FUNCTION FC_InitRaInterface : BOOL
VAR_INPUT
END_VAR
VAR
	i: UINT;
	m_statesEnum: EProcessVariables;
END_VAR

// OUT - alarms
FOR i := ResiConst.ARR_MIN TO RaInterface_GVL.ALARM_ARR_MAX DO
	RaInterface_GVL.Out_Alarms[i].Active := FALSE;
	RaInterface_GVL.Out_Alarms[i].AlarmId := 0;
	RaInterface_GVL.Out_Alarms[i].InstanceName := '';
	RaInterface_GVL.Out_Alarms[i].Message := '';
	RaInterface_GVL.Out_Alarms[i].Severity := ESeverity.none;
	RaInterface_GVL.Out_Alarms[i].TimeTicks := 0;
END_FOR

// OUT - process state
FOR i := ResiConst.ARR_MIN TO ResiConst.STATE_ARR_MAX DO
	m_statesEnum := i;
	RaInterface_GVL.Out_NamedProcessState[i].Name := TO_STRING(m_statesEnum);
END_FOR

// OUT - recovery request
RaInterface_GVL.Out_RecoveryRequest.ChangeTrigger := 0;
RaInterface_GVL.Out_RecoveryRequest.RequestedState := '';

END_FUNCTION

(* stored: Version 1.1.0.1, ProductVersion 3.1.4024.9
   POU FC_InitRaInterface: Id {b6ec912e-68c2-4707-bca3-802686777af9}, SpecialFunc None *)
